FUNCTION_BLOCK FB_SmokeDetector EXTENDS FB_BaseSensor
VAR_INPUT
END_VAR
VAR_OUTPUT
END_VAR
VAR
END_VAR

// Handle fault simulation
IF bSimFault THEN
    _bFault  := TRUE;
    _eStatus := E_SensorStatus.SENSOR_FAULT;
    RETURN;
END_IF

// Accept raw value
_rValue := rRawValue;

// Call abstract validate — child implements this
THIS^.Validate();

METHOD  Validate 
VAR_INPUT
END_VAR
// Smoke detector is binary — any reading above 0 is alarm
// rRawValue: 0.0 = clear, 1.0 = smoke detected
IF _rValue < 0.0 OR _rValue > 1.0 THEN
    _bFault  := TRUE;
    _eStatus := E_SensorStatus.SENSOR_FAULT;
    RETURN;
END_IF

IF _rValue >= 1.0 THEN
    _bAlarm  := TRUE;
    _eStatus := E_SensorStatus.SENSOR_ALARM;
ELSE
    _bAlarm  := FALSE;
    _eStatus := E_SensorStatus.SENSOR_OK;
END_IF
END_METHOD

END_FUNCTION_BLOCK

(* stored: Version 1.1.0.1, ProductVersion 3.1.4024.16
   POU FB_SmokeDetector: Id {9852d6d9-667c-4618-b34f-5dd8fa55f0a6}, SpecialFunc None
   Method Validate: Id {d085ccb5-43bb-45d4-9bd9-fbd98c3b9594} *)
